TYPE ST_Camera_CMD :
STRUCT
	
	Extend				: BOOL;		
	Retract				: BOOL;		
	
END_STRUCT
END_TYPE

(* stored: Version 1.1.0.1, ProductVersion 3.1.4024.13
   DUT ST_Camera_CMD: Id {b04f1e4d-e0a9-4657-bf3c-f43eae8c4118} *)
